FUNCTION_BLOCK FB_OR_3 (* Boolean OR *)
  (* Standard: 61499-1-D.1; Classification: Boolean functions *)
  (* Version 0.1, 2001-08-05, JHC, Rockwell Automation, XML version *)
  (* Version 0.0, 2000-01-10, JHC, Rockwell Automation, SRC version *)
  (* Compiler header: package fb.rt.student; *)
  (* Compiler classdef: class FB_OR extends FBFunction2 *)
  (* Compiler Java IBM VisualAge 3.0 *)
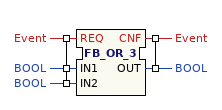
  EVENT_INPUT
    REQ WITH IN1, IN2;
  END_EVENT
  EVENT_OUTPUT
    CNF WITH OUT;
  END_EVENT
  VAR_INPUT
    IN1 : BOOL;
    IN2 : BOOL;
  END_VAR
  VAR_OUTPUT
    OUT : BOOL; (* Result *)
  END_VAR
END_FUNCTION_BLOCK
